TYPE ST_Test :
STRUCT
	var1: BOOL;
	var2: INT;
	VarArray: ARRAY [0..11] OF INT;
END_STRUCT
END_TYPE

(* stored: Version 1.1.0.1, ProductVersion 3.1.4024.6
   DUT ST_Test: Id {6bcd14f4-0128-41bb-b0cd-471b9f79867c} *)
